TYPE E_CtrlId :
(
	//not defined after startup...
	NONE,
	RFW_11,
	CYL_1,
	VPC_1,	
	UMC_1,	
	PRS_1,	
	BCC_1,
	DRV_1,
	RFW_12,
	ACL_1,
	VLV_1,
	ECD_1,
	E_CtrlIdMax
);
END_TYPE

(* stored: Version 1.1.0.1, ProductVersion 3.1.0.23
   DUT E_CtrlId: Id {fbb9f2d2-c911-4ba8-bff4-7e84f684cb30} *)
